KUKA KRL program: chk_w5_wechs_ok.src

&ACCESS RVO7
&REL 1
&COMMENT Check Pinca Axor
DEF chk_w5_wechs_ok( )

; VERIFICAÇÃO DE FERRAMENTE: PINCA AXOR/ATEGO

WAIT FOR (($in[161]) AND ($in[169]) AND  ($in[177]) AND ($in[185]) AND (NOT $in[193]) AND (($IN[201]) OR ((NOT $IN[201]) AND ($IN [3320]))) AND ($in[219]))

END
